PROGRAM PRG_AssignValToStringWithPrefixManual
VAR
	asRejectReason		: T_MaxString;
	anValue				: ARRAY[0..10] OF STRING(10);
	asPointer          	: ARRAY[0..10] OF STRING(10);
	nPrefixSize			: UINT;
	nPrefixValue		: STRING(5);
	
	F_AssignValToStringWithPrefix	: T_MaxString;
	
	//from FFB_CASE_DuplicatCheck - outer duplicate
	nDuplicateOuter1_Position		: INT;
	nDuplicateOuter2_Position		: INT;
	

END_VAR

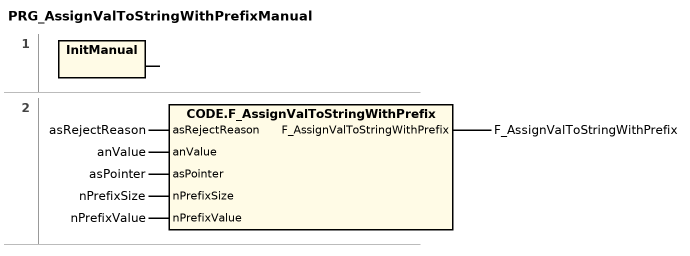
// NETWORK 1
InitManual();

// NETWORK 2
F_AssignValToStringWithPrefix := CODE.F_AssignValToStringWithPrefix(asRejectReason := asRejectReason, anValue := anValue, asPointer := asPointer, nPrefixSize := nPrefixSize, nPrefixValue := nPrefixValue);

ACTION InitManual:

asRejectReason := 'XXINVnnXX';

nPrefixSize	 := 2;
nPrefixValue := '0' ;

asPointer[0] := 'nn';
asPointer[1] := 'n2';

nDuplicateOuter1_Position := 2;
nDuplicateOuter2_Position := 4;

//anValue[0] := 	F_StringAddPrefix(INT_TO_STRING(nDuplicateOuter1_Position),2,'0');
//anValue[1] := 	F_StringAddPrefix(INT_TO_STRING(nDuplicateOuter2_Position),2,'0');

anValue[0] := TO_STRING(nDuplicateOuter1_Position);
anValue[1] := TO_STRING(nDuplicateOuter2_Position);
END_ACTION

END_PROGRAM

(* stored: Version 1.1.0.1
   POU PRG_AssignValToStringWithPrefixManual: Id {40a84d3c-0d1d-46ca-b11a-27e190de3ddf}, SpecialFunc None
   Action InitManual: Id {af4fa378-0741-4677-b846-ff59ad3bb584} *)
